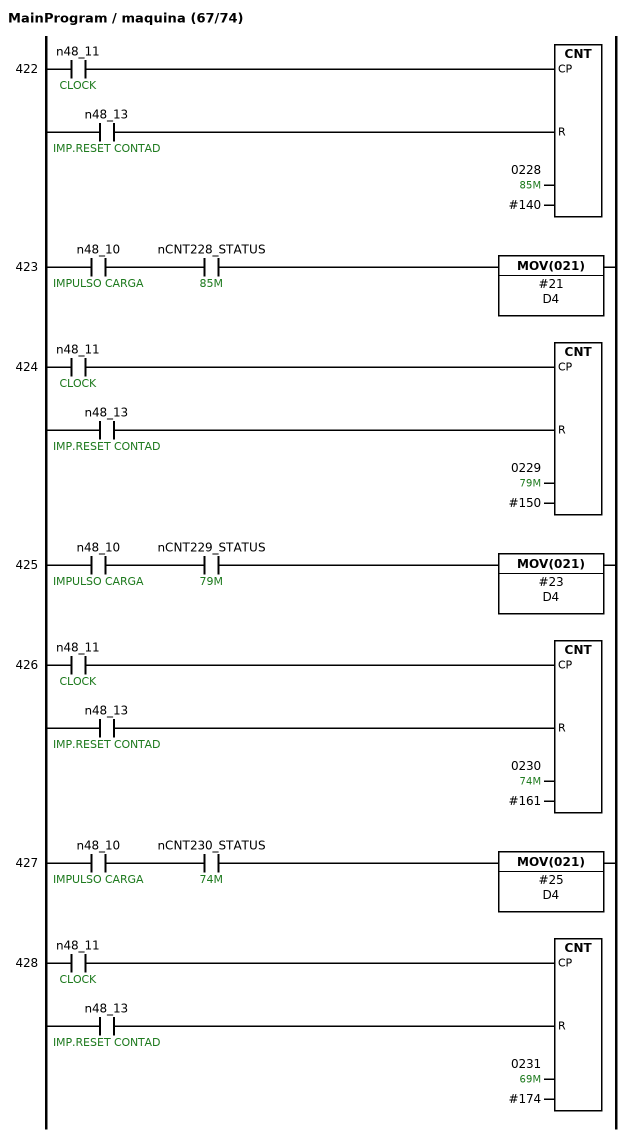
; [picture p72: MainProgram / maquina, rungs 422-428]
; rung 422
LD n48_11  ; CLOCK
LD n48_13  ; IMP.RESET CONTAD
CNT 0228 #140  ; 85M
; rung 423
LD n48_10  ; IMPULSO CARGA
AND nCNT228_STATUS  ; 85M
MOV(021) #21 D4
; rung 424
LD n48_11  ; CLOCK
LD n48_13  ; IMP.RESET CONTAD
CNT 0229 #150  ; 79M
; rung 425
LD n48_10  ; IMPULSO CARGA
AND nCNT229_STATUS  ; 79M
MOV(021) #23 D4
; rung 426
LD n48_11  ; CLOCK
LD n48_13  ; IMP.RESET CONTAD
CNT 0230 #161  ; 74M
; rung 427
LD n48_10  ; IMPULSO CARGA
AND nCNT230_STATUS  ; 74M
MOV(021) #25 D4
; rung 428
LD n48_11  ; CLOCK
LD n48_13  ; IMP.RESET CONTAD
CNT 0231 #174  ; 69M

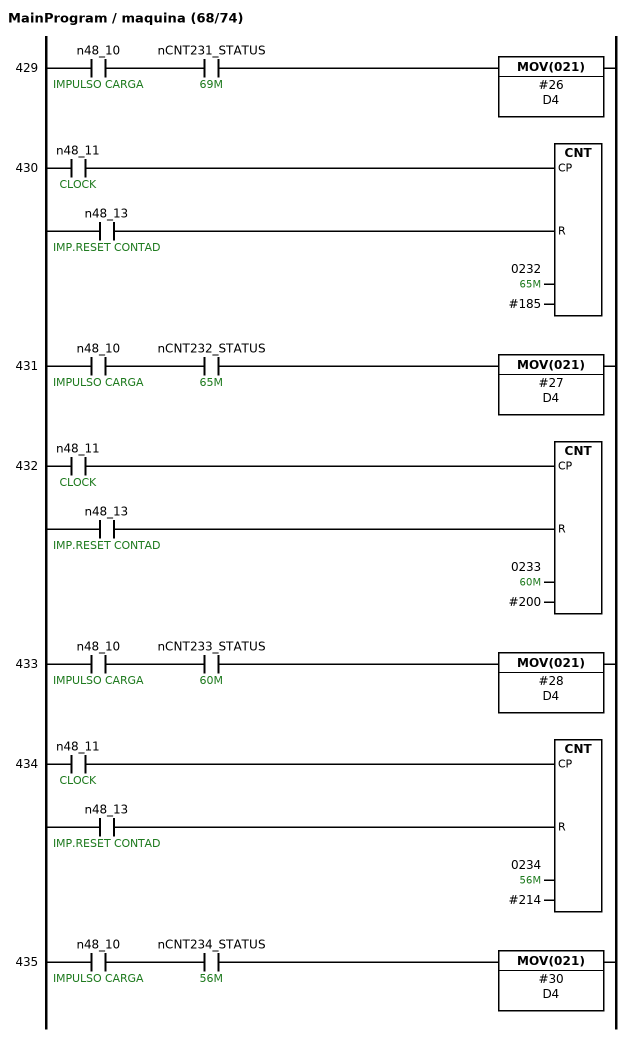
; rung 429
LD n48_10  ; IMPULSO CARGA
AND nCNT231_STATUS  ; 69M
MOV(021) #26 D4
; rung 430
LD n48_11  ; CLOCK
LD n48_13  ; IMP.RESET CONTAD
CNT 0232 #185  ; 65M
; rung 431
LD n48_10  ; IMPULSO CARGA
AND nCNT232_STATUS  ; 65M
MOV(021) #27 D4
; rung 432
LD n48_11  ; CLOCK
LD n48_13  ; IMP.RESET CONTAD
CNT 0233 #200  ; 60M
; rung 433
LD n48_10  ; IMPULSO CARGA
AND nCNT233_STATUS  ; 60M
MOV(021) #28 D4
; rung 434
LD n48_11  ; CLOCK
LD n48_13  ; IMP.RESET CONTAD
CNT 0234 #214  ; 56M
; rung 435
LD n48_10  ; IMPULSO CARGA
AND nCNT234_STATUS  ; 56M
MOV(021) #30 D4

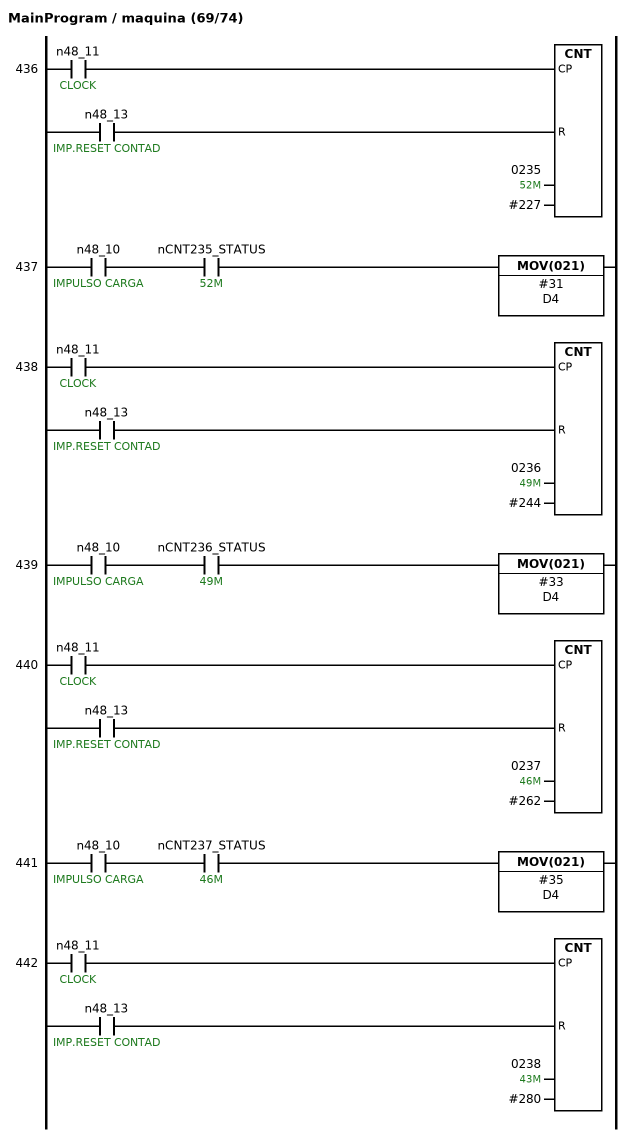
; rung 436
LD n48_11  ; CLOCK
LD n48_13  ; IMP.RESET CONTAD
CNT 0235 #227  ; 52M
; rung 437
LD n48_10  ; IMPULSO CARGA
AND nCNT235_STATUS  ; 52M
MOV(021) #31 D4
; rung 438
LD n48_11  ; CLOCK
LD n48_13  ; IMP.RESET CONTAD
CNT 0236 #244  ; 49M
; rung 439
LD n48_10  ; IMPULSO CARGA
AND nCNT236_STATUS  ; 49M
MOV(021) #33 D4
; rung 440
LD n48_11  ; CLOCK
LD n48_13  ; IMP.RESET CONTAD
CNT 0237 #262  ; 46M
; rung 441
LD n48_10  ; IMPULSO CARGA
AND nCNT237_STATUS  ; 46M
MOV(021) #35 D4
; rung 442
LD n48_11  ; CLOCK
LD n48_13  ; IMP.RESET CONTAD
CNT 0238 #280  ; 43M

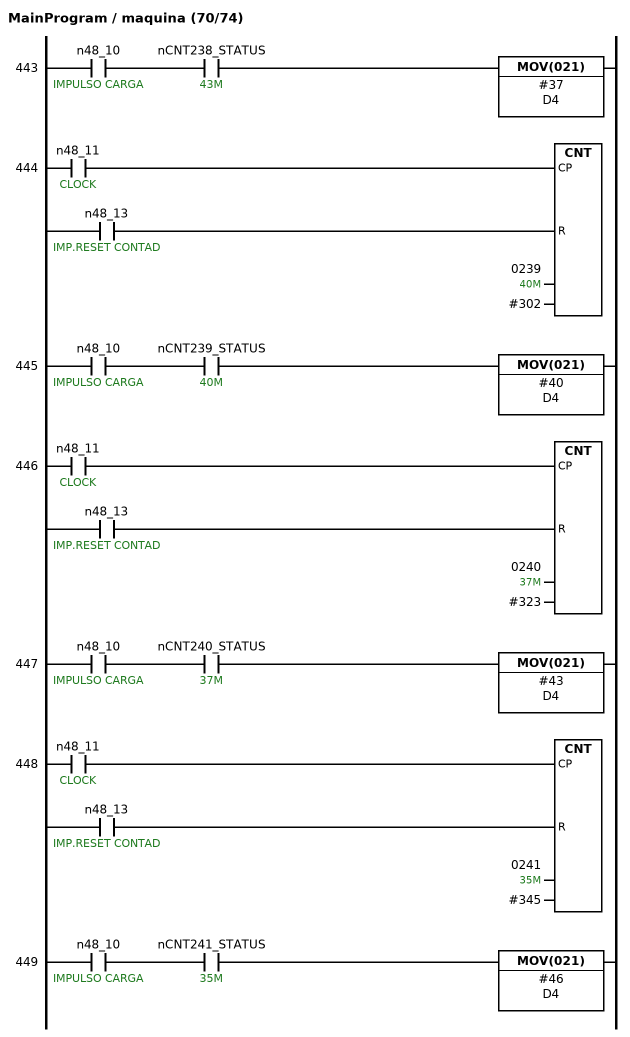
; rung 443
LD n48_10  ; IMPULSO CARGA
AND nCNT238_STATUS  ; 43M
MOV(021) #37 D4
; rung 444
LD n48_11  ; CLOCK
LD n48_13  ; IMP.RESET CONTAD
CNT 0239 #302  ; 40M
; rung 445
LD n48_10  ; IMPULSO CARGA
AND nCNT239_STATUS  ; 40M
MOV(021) #40 D4
; rung 446
LD n48_11  ; CLOCK
LD n48_13  ; IMP.RESET CONTAD
CNT 0240 #323  ; 37M
; rung 447
LD n48_10  ; IMPULSO CARGA
AND nCNT240_STATUS  ; 37M
MOV(021) #43 D4
; rung 448
LD n48_11  ; CLOCK
LD n48_13  ; IMP.RESET CONTAD
CNT 0241 #345  ; 35M
; rung 449
LD n48_10  ; IMPULSO CARGA
AND nCNT241_STATUS  ; 35M
MOV(021) #46 D4

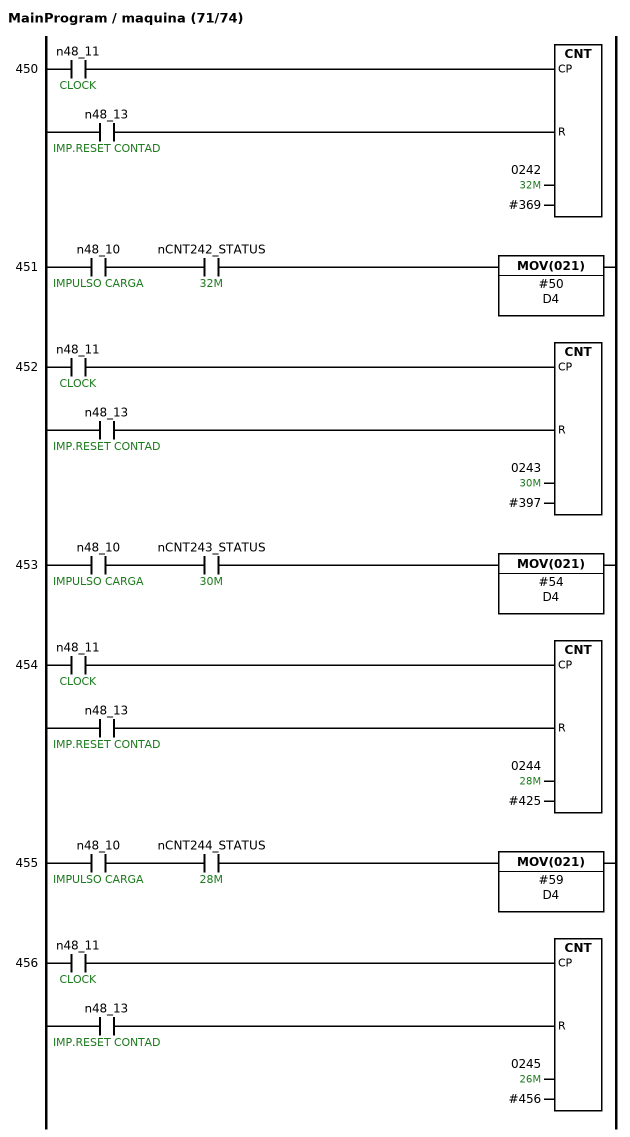
; rung 450
LD n48_11  ; CLOCK
LD n48_13  ; IMP.RESET CONTAD
CNT 0242 #369  ; 32M
; rung 451
LD n48_10  ; IMPULSO CARGA
AND nCNT242_STATUS  ; 32M
MOV(021) #50 D4
; rung 452
LD n48_11  ; CLOCK
LD n48_13  ; IMP.RESET CONTAD
CNT 0243 #397  ; 30M
; rung 453
LD n48_10  ; IMPULSO CARGA
AND nCNT243_STATUS  ; 30M
MOV(021) #54 D4
; rung 454
LD n48_11  ; CLOCK
LD n48_13  ; IMP.RESET CONTAD
CNT 0244 #425  ; 28M
; rung 455
LD n48_10  ; IMPULSO CARGA
AND nCNT244_STATUS  ; 28M
MOV(021) #59 D4
; rung 456
LD n48_11  ; CLOCK
LD n48_13  ; IMP.RESET CONTAD
CNT 0245 #456  ; 26M

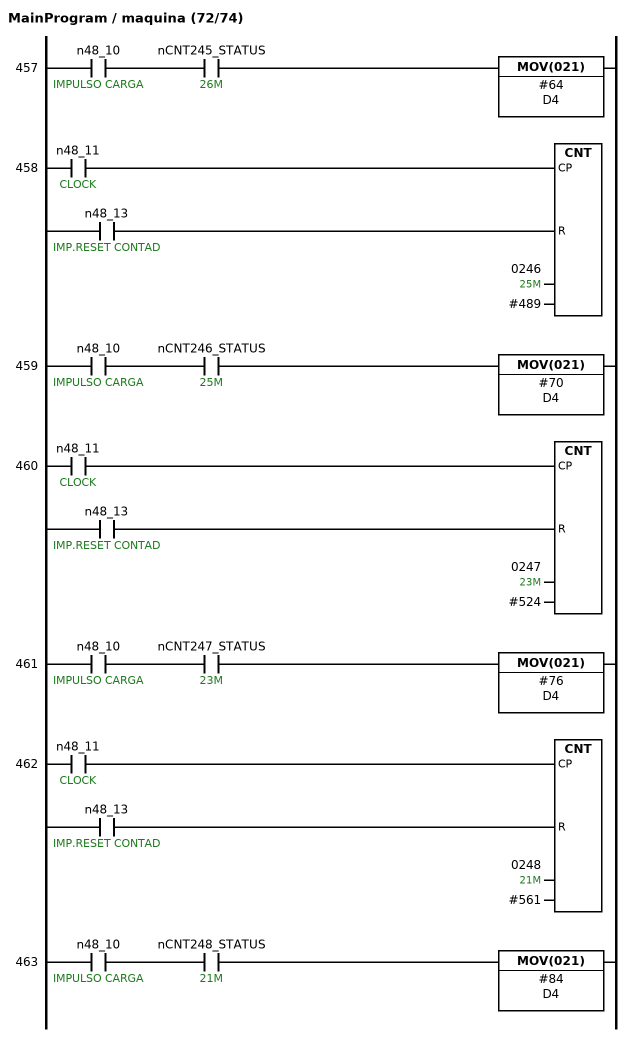
; rung 457
LD n48_10  ; IMPULSO CARGA
AND nCNT245_STATUS  ; 26M
MOV(021) #64 D4
; rung 458
LD n48_11  ; CLOCK
LD n48_13  ; IMP.RESET CONTAD
CNT 0246 #489  ; 25M
; rung 459
LD n48_10  ; IMPULSO CARGA
AND nCNT246_STATUS  ; 25M
MOV(021) #70 D4
; rung 460
LD n48_11  ; CLOCK
LD n48_13  ; IMP.RESET CONTAD
CNT 0247 #524  ; 23M
; rung 461
LD n48_10  ; IMPULSO CARGA
AND nCNT247_STATUS  ; 23M
MOV(021) #76 D4
; rung 462
LD n48_11  ; CLOCK
LD n48_13  ; IMP.RESET CONTAD
CNT 0248 #561  ; 21M
; rung 463
LD n48_10  ; IMPULSO CARGA
AND nCNT248_STATUS  ; 21M
MOV(021) #84 D4

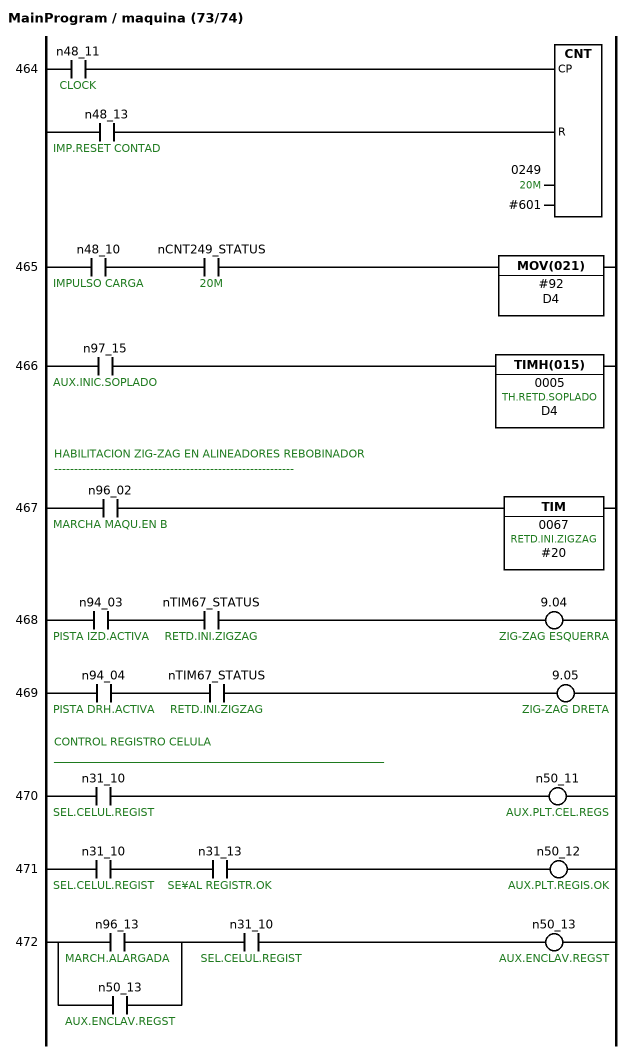
; rung 464
LD n48_11  ; CLOCK
LD n48_13  ; IMP.RESET CONTAD
CNT 0249 #601  ; 20M
; rung 465
LD n48_10  ; IMPULSO CARGA
AND nCNT249_STATUS  ; 20M
MOV(021) #92 D4
; rung 466
LD n97_15  ; AUX.INIC.SOPLADO
TIMH(015) 0005 D4  ; TH.RETD.SOPLADO
; rung 467: HABILITACION ZIG-ZAG EN ALINEADORES REBOBINADOR / ------------------------------------------------------------
LD n96_02  ; MARCHA MAQU.EN B
TIM 0067 #20  ; RETD.INI.ZIGZAG
; rung 468
LD n94_03  ; PISTA IZD.ACTIVA
AND nTIM67_STATUS  ; RETD.INI.ZIGZAG
OUT 9.04  ; ZIG-ZAG ESQUERRA
; rung 469
LD n94_04  ; PISTA DRH.ACTIVA
AND nTIM67_STATUS  ; RETD.INI.ZIGZAG
OUT 9.05  ; ZIG-ZAG DRETA
; rung 470: CONTROL REGISTRO CELULA / ____________________________________________________________
LD n31_10  ; SEL.CELUL.REGIST
OUT n50_11  ; AUX.PLT.CEL.REGS
; rung 471
LD n31_10  ; SEL.CELUL.REGIST
AND n31_13  ; SE¥AL REGISTR.OK
OUT n50_12  ; AUX.PLT.REGIS.OK
; rung 472
LD n96_13  ; MARCH.ALARGADA
OR n50_13  ; AUX.ENCLAV.REGST
AND n31_10  ; SEL.CELUL.REGIST
OUT n50_13  ; AUX.ENCLAV.REGST

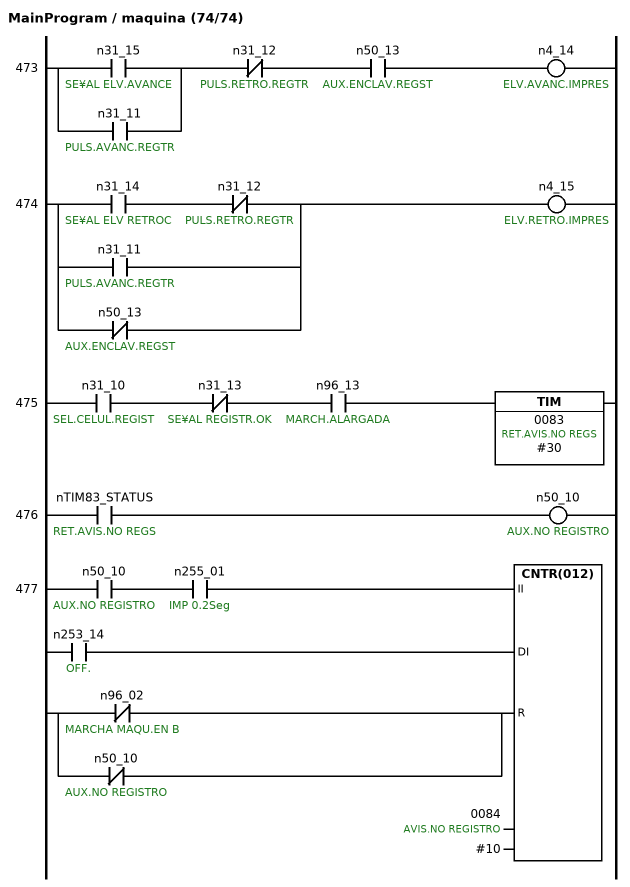
; rung 473
LD n31_15  ; SE¥AL ELV.AVANCE
OR n31_11  ; PULS.AVANC.REGTR
ANDNOT n31_12  ; PULS.RETRO.REGTR
AND n50_13  ; AUX.ENCLAV.REGST
OUT n4_14  ; ELV.AVANC.IMPRES
; rung 474
LD n31_14  ; SE¥AL ELV RETROC
ANDNOT n31_12  ; PULS.RETRO.REGTR
OR n31_11  ; PULS.AVANC.REGTR
ORNOT n50_13  ; AUX.ENCLAV.REGST
OUT n4_15  ; ELV.RETRO.IMPRES
; rung 475
LD n31_10  ; SEL.CELUL.REGIST
ANDNOT n31_13  ; SE¥AL REGISTR.OK
AND n96_13  ; MARCH.ALARGADA
TIM 0083 #30  ; RET.AVIS.NO REGS
; rung 476
LD nTIM83_STATUS  ; RET.AVIS.NO REGS
OUT n50_10  ; AUX.NO REGISTRO
; rung 477
LD n50_10  ; AUX.NO REGISTRO
AND n255_01  ; IMP 0.2Seg
LD n253_14  ; OFF.
LDNOT n96_02  ; MARCHA MAQU.EN B
ORNOT n50_10  ; AUX.NO REGISTRO
CNTR(012) 0084 #10  ; AVIS.NO REGISTRO

### Section Aliniadors

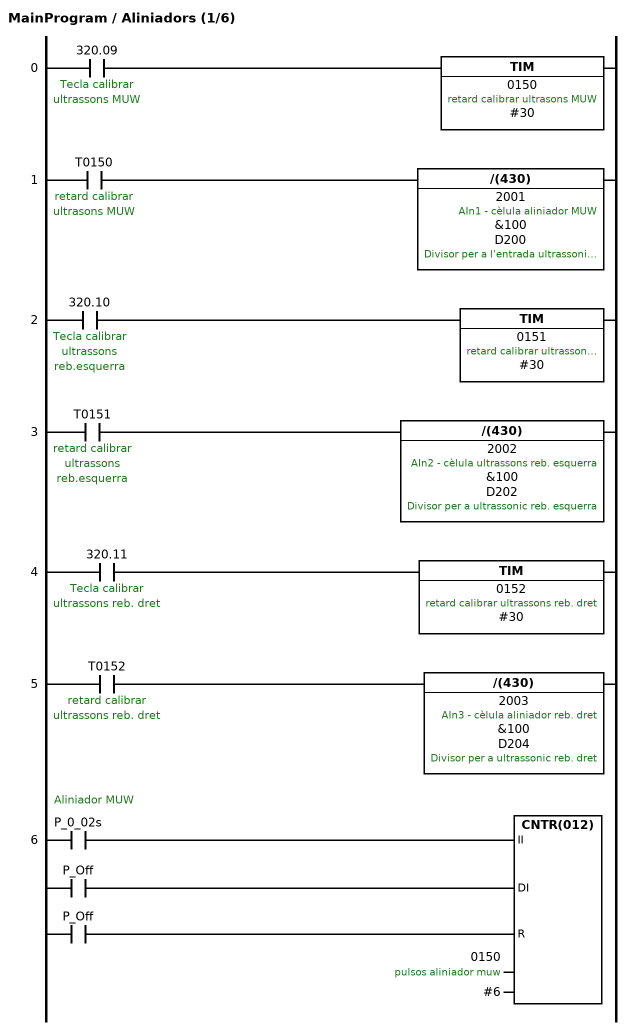
; rung 0
LD 320.09  ; Tecla calibrar ultrassons MUW
TIM 0150 #30  ; retard calibrar ultrasons MUW
; rung 1
LD T0150  ; retard calibrar ultrasons MUW
/(430) 2001 &100 D200  ; AIn1 - cèlula aliniador MUW, Divisor per a l'entrada ultrassonic MUW
; rung 2
LD 320.10  ; Tecla calibrar ultrassons reb.esquerra
TIM 0151 #30  ; retard calibrar ultrassons reb.esquerra
; rung 3
LD T0151  ; retard calibrar ultrassons reb.esquerra
/(430) 2002 &100 D202  ; AIn2 - cèlula ultrassons reb. esquerra, Divisor per a ultrassonic reb. esquerra
; rung 4
LD 320.11  ; Tecla calibrar ultrassons reb. dret
TIM 0152 #30  ; retard calibrar ultrassons reb. dret
; rung 5
LD T0152  ; retard calibrar ultrassons reb. dret
/(430) 2003 &100 D204  ; AIn3 - cèlula aliniador reb. dret, Divisor per a ultrassonic reb. dret
; rung 6: Aliniador MUW
LD P_0_02s
LD P_Off
LD P_Off
CNTR(012) 0150 #6  ; pulsos aliniador muw

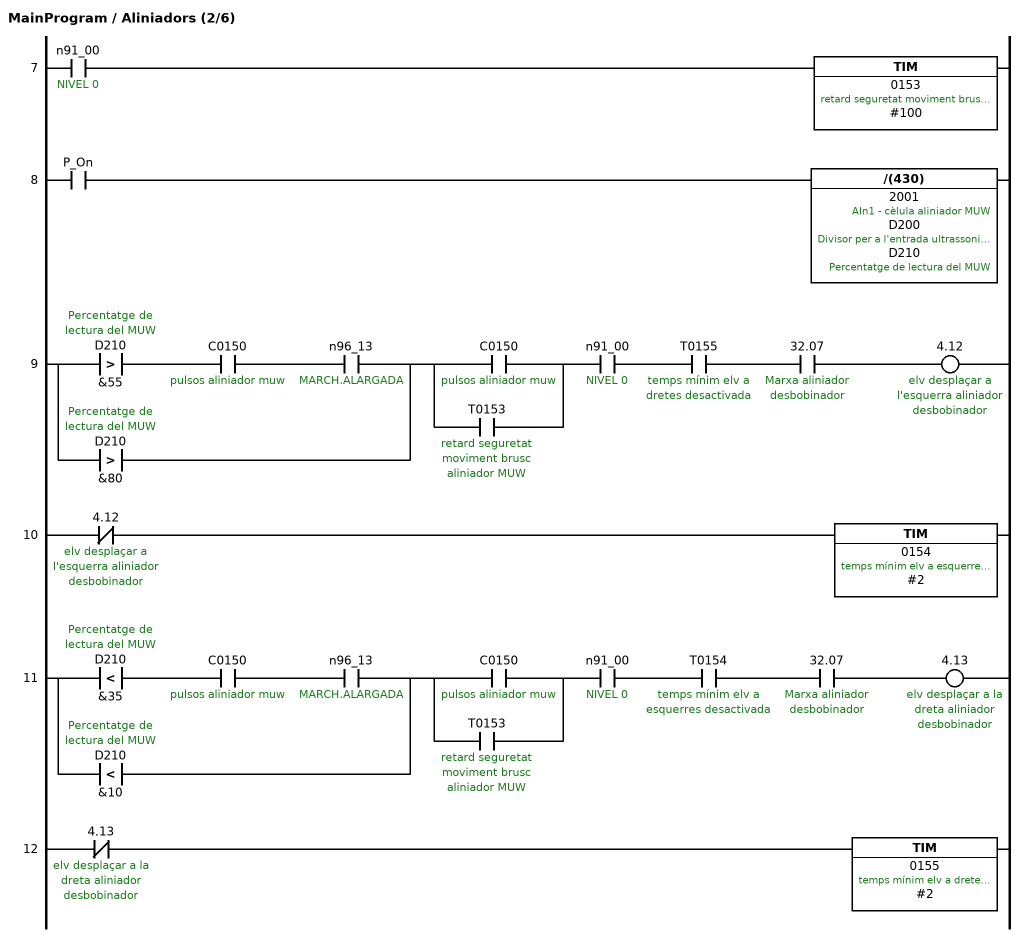
; rung 7
LD n91_00  ; NIVEL 0
TIM 0153 #100  ; retard seguretat moviment brusc aliniador MUW
; rung 8
LD P_On
/(430) 2001 D200 D210  ; AIn1 - cèlula aliniador MUW, Divisor per a l'entrada ultrassonic MUW, Percentatge de lectura del MUW
; rung 9
LD>(320) D210 &55  ; Percentatge de lectura del MUW
AND C0150  ; pulsos aliniador muw
AND n96_13  ; MARCH.ALARGADA
OR>(320) D210 &80  ; Percentatge de lectura del MUW
LD C0150  ; pulsos aliniador muw
OR T0153  ; retard seguretat moviment brusc aliniador MUW
ANDLD
AND n91_00  ; NIVEL 0
AND T0155  ; temps mínim elv a dretes desactivada
AND 32.07  ; Marxa aliniador desbobinador
OUT 4.12  ; elv desplaçar a l'esquerra aliniador desbobinador
; rung 10
LDNOT 4.12  ; elv desplaçar a l'esquerra aliniador desbobinador
TIM 0154 #2  ; temps mínim elv a esquerres desactivada
; rung 11
LD<(310) D210 &35  ; Percentatge de lectura del MUW
AND C0150  ; pulsos aliniador muw
AND n96_13  ; MARCH.ALARGADA
OR<(310) D210 &10  ; Percentatge de lectura del MUW
LD C0150  ; pulsos aliniador muw
OR T0153  ; retard seguretat moviment brusc aliniador MUW
ANDLD
AND n91_00  ; NIVEL 0
AND T0154  ; temps mínim elv a esquerres desactivada
AND 32.07  ; Marxa aliniador desbobinador
OUT 4.13  ; elv desplaçar a la dreta aliniador desbobinador
; rung 12
LDNOT 4.13  ; elv desplaçar a la dreta aliniador desbobinador
TIM 0155 #2  ; temps mínim elv a dretes desactivada

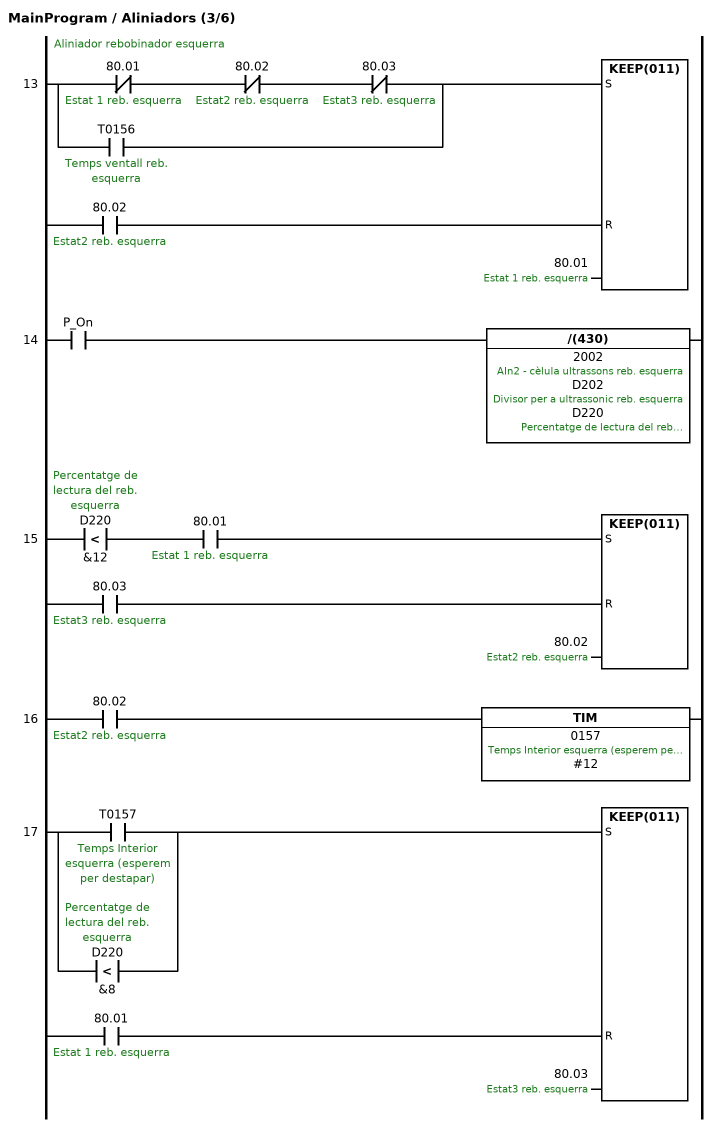
; rung 13: Aliniador rebobinador esquerra
LDNOT 80.01  ; Estat 1 reb. esquerra
ANDNOT 80.02  ; Estat2 reb. esquerra
ANDNOT 80.03  ; Estat3 reb. esquerra
OR T0156  ; Temps ventall reb. esquerra
LD 80.02  ; Estat2 reb. esquerra
KEEP(011) 80.01  ; Estat 1 reb. esquerra
; rung 14
LD P_On
/(430) 2002 D202 D220  ; AIn2 - cèlula ultrassons reb. esquerra, Divisor per a ultrassonic reb. esquerra, Percentatge de lectura del reb. esquerra
; rung 15
LD<(310) D220 &12  ; Percentatge de lectura del reb. esquerra
AND 80.01  ; Estat 1 reb. esquerra
LD 80.03  ; Estat3 reb. esquerra
KEEP(011) 80.02  ; Estat2 reb. esquerra
; rung 16
LD 80.02  ; Estat2 reb. esquerra
TIM 0157 #12  ; Temps Interior esquerra (esperem per destapar)
; rung 17
LD T0157  ; Temps Interior esquerra (esperem per destapar)
OR<(310) D220 &8  ; Percentatge de lectura del reb. esquerra
LD 80.01  ; Estat 1 reb. esquerra
KEEP(011) 80.03  ; Estat3 reb. esquerra

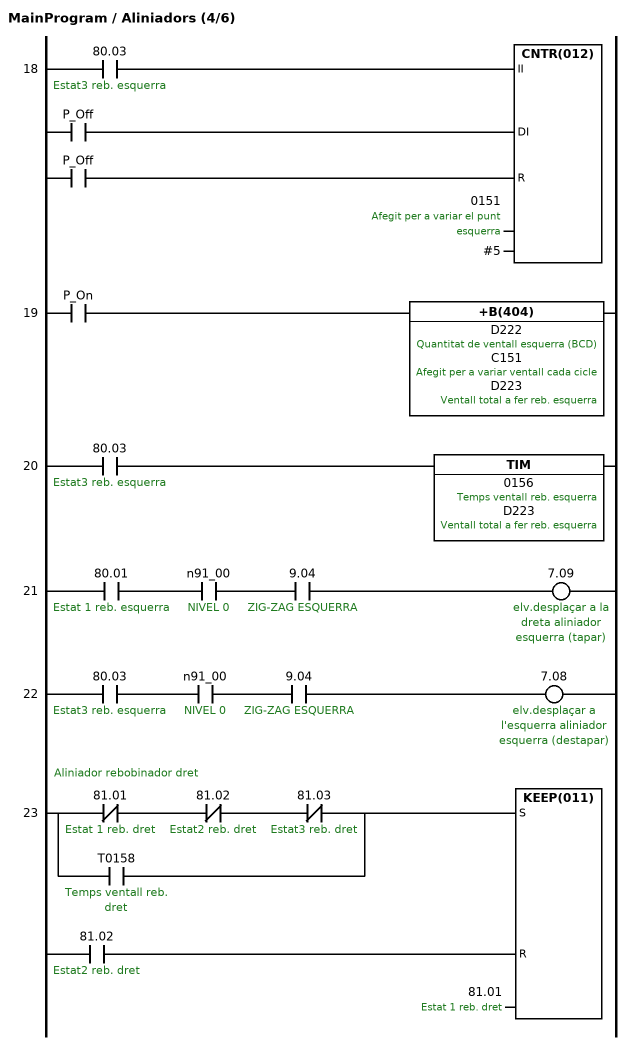
; rung 18
LD 80.03  ; Estat3 reb. esquerra
LD P_Off
LD P_Off
CNTR(012) 0151 #5  ; Afegit per a variar el punt esquerra
; rung 19
LD P_On
+B(404) D222 C151 D223  ; Quantitat de ventall esquerra (BCD), Afegit per a variar ventall cada cicle, Ventall total a fer reb. esquerra
; rung 20
LD 80.03  ; Estat3 reb. esquerra
TIM 0156 D223  ; Ventall total a fer reb. esquerra, Temps ventall reb. esquerra
; rung 21
LD 80.01  ; Estat 1 reb. esquerra
AND n91_00  ; NIVEL 0
AND 9.04  ; ZIG-ZAG ESQUERRA
OUT 7.09  ; elv.desplaçar a la dreta aliniador esquerra (tapar)
; rung 22
LD 80.03  ; Estat3 reb. esquerra
AND n91_00  ; NIVEL 0
AND 9.04  ; ZIG-ZAG ESQUERRA
OUT 7.08  ; elv.desplaçar a l'esquerra aliniador esquerra (destapar)
; rung 23: Aliniador rebobinador dret
LDNOT 81.01  ; Estat 1 reb. dret
ANDNOT 81.02  ; Estat2 reb. dret
ANDNOT 81.03  ; Estat3 reb. dret
OR T0158  ; Temps ventall reb. dret
LD 81.02  ; Estat2 reb. dret
KEEP(011) 81.01  ; Estat 1 reb. dret

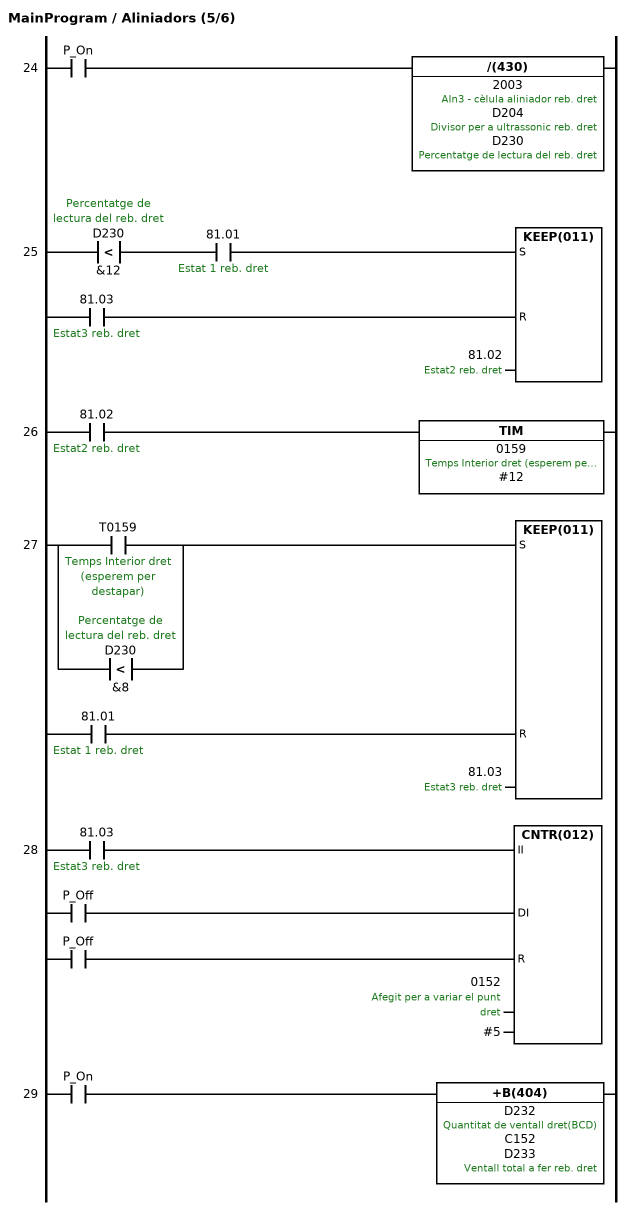
; rung 24
LD P_On
/(430) 2003 D204 D230  ; AIn3 - cèlula aliniador reb. dret, Divisor per a ultrassonic reb. dret, Percentatge de lectura del reb. dret
; rung 25
LD<(310) D230 &12  ; Percentatge de lectura del reb. dret
AND 81.01  ; Estat 1 reb. dret
LD 81.03  ; Estat3 reb. dret
KEEP(011) 81.02  ; Estat2 reb. dret
; rung 26
LD 81.02  ; Estat2 reb. dret
TIM 0159 #12  ; Temps Interior dret (esperem per destapar)
; rung 27
LD T0159  ; Temps Interior dret (esperem per destapar)
OR<(310) D230 &8  ; Percentatge de lectura del reb. dret
LD 81.01  ; Estat 1 reb. dret
KEEP(011) 81.03  ; Estat3 reb. dret
; rung 28
LD 81.03  ; Estat3 reb. dret
LD P_Off
LD P_Off
CNTR(012) 0152 #5  ; Afegit per a variar el punt dret
; rung 29
LD P_On
+B(404) D232 C152 D233  ; Quantitat de ventall dret(BCD), Ventall total a fer reb. dret

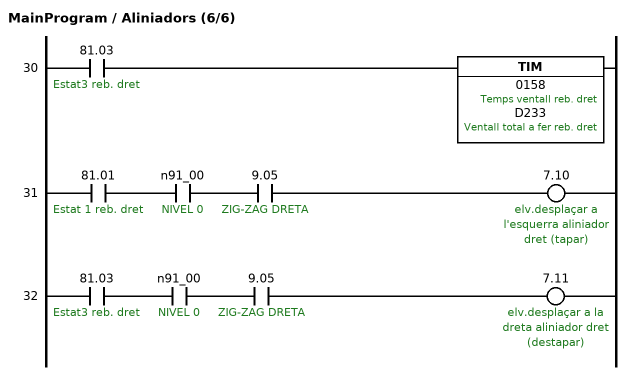
; rung 30
LD 81.03  ; Estat3 reb. dret
TIM 0158 D233  ; Ventall total a fer reb. dret, Temps ventall reb. dret
; rung 31
LD 81.01  ; Estat 1 reb. dret
AND n91_00  ; NIVEL 0
AND 9.05  ; ZIG-ZAG DRETA
OUT 7.10  ; elv.desplaçar a l'esquerra aliniador dret (tapar)
; rung 32
LD 81.03  ; Estat3 reb. dret
AND n91_00  ; NIVEL 0
AND 9.05  ; ZIG-ZAG DRETA
OUT 7.11  ; elv.desplaçar a la dreta aliniador dret (destapar)

### Section HMI

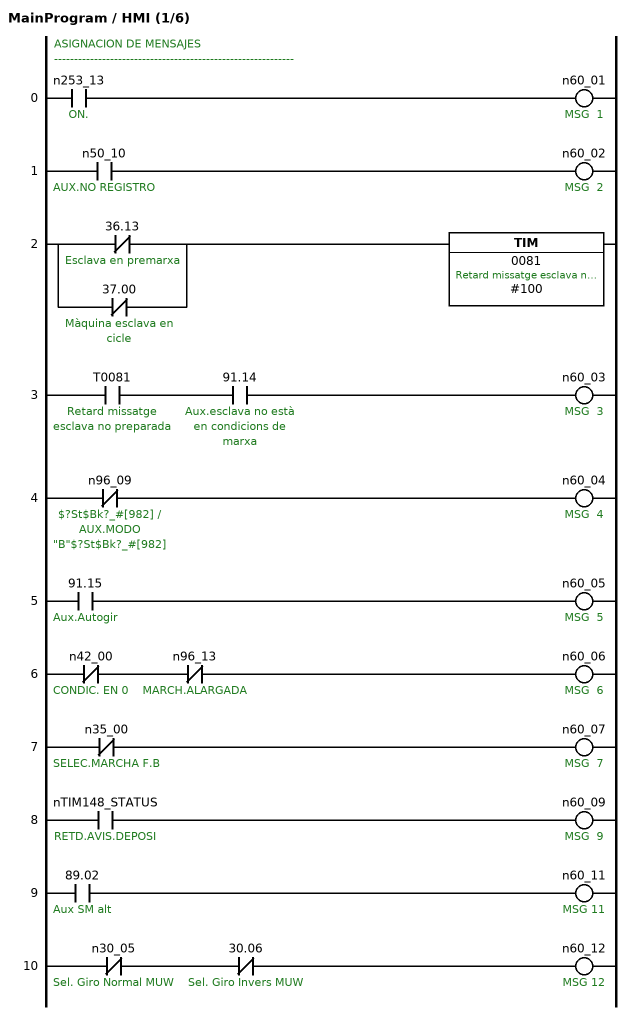
; rung 0: ASIGNACION DE MENSAJES / ------------------------------------------------------------
LD n253_13  ; ON.
OUT n60_01  ; MSG  1
; rung 1
LD n50_10  ; AUX.NO REGISTRO
OUT n60_02  ; MSG  2
; rung 2
LDNOT 36.13  ; Esclava en premarxa
ORNOT 37.00  ; Màquina esclava en cicle
TIM 0081 #100  ; Retard missatge esclava no preparada
; rung 3
LD T0081  ; Retard missatge esclava no preparada
AND 91.14  ; Aux.esclava no està en condicions de marxa
OUT n60_03  ; MSG  3
; rung 4
LDNOT n96_09  ; $?St$Bk?_#[982] / AUX.MODO "B"$?St$Bk?_#[982]
OUT n60_04  ; MSG  4
; rung 5
LD 91.15  ; Aux.Autogir
OUT n60_05  ; MSG  5
; rung 6
LDNOT n42_00  ; CONDIC. EN 0
ANDNOT n96_13  ; MARCH.ALARGADA
OUT n60_06  ; MSG  6
; rung 7
LDNOT n35_00  ; SELEC.MARCHA F.B
OUT n60_07  ; MSG  7
; rung 8
LD nTIM148_STATUS  ; RETD.AVIS.DEPOSI
OUT n60_09  ; MSG  9
; rung 9
LD 89.02  ; Aux SM alt
OUT n60_11  ; MSG 11
; rung 10
LDNOT n30_05  ; Sel. Giro Normal MUW
ANDNOT 30.06  ; Sel. Giro Invers MUW
OUT n60_12  ; MSG 12

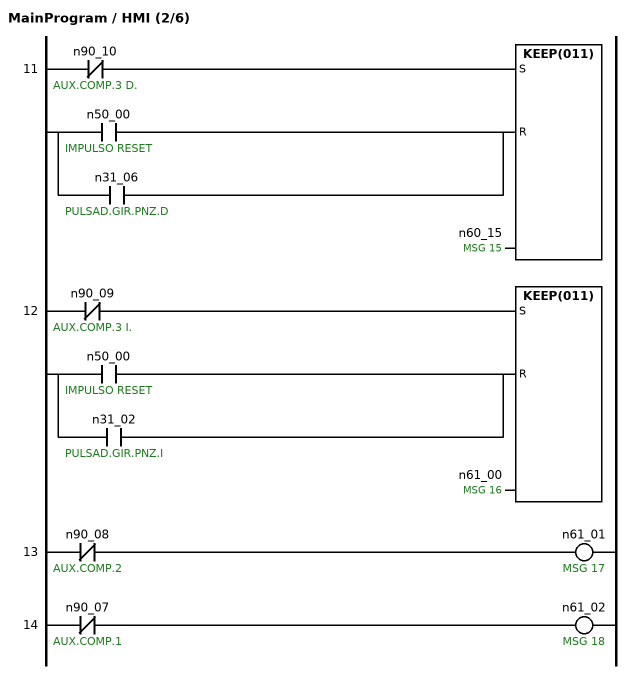
; rung 11
LDNOT n90_10  ; AUX.COMP.3 D.
LD n50_00  ; IMPULSO RESET
OR n31_06  ; PULSAD.GIR.PNZ.D
KEEP(011) n60_15  ; MSG 15
; rung 12
LDNOT n90_09  ; AUX.COMP.3 I.
LD n50_00  ; IMPULSO RESET
OR n31_02  ; PULSAD.GIR.PNZ.I
KEEP(011) n61_00  ; MSG 16
; rung 13
LDNOT n90_08  ; AUX.COMP.2
OUT n61_01  ; MSG 17
; rung 14
LDNOT n90_07  ; AUX.COMP.1
OUT n61_02  ; MSG 18

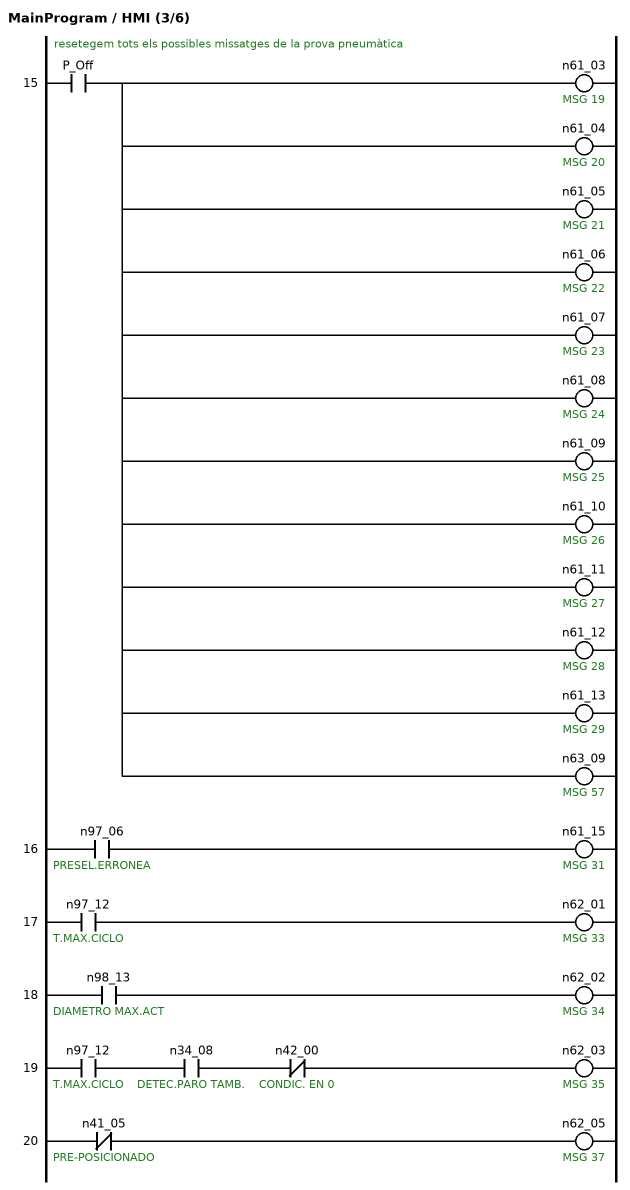
; rung 15: resetegem tots els possibles missatges de la prova pneumàtica
LD P_Off
OUT n61_03  ; MSG 19
OUT n61_04  ; MSG 20
OUT n61_05  ; MSG 21
OUT n61_06  ; MSG 22
OUT n61_07  ; MSG 23
OUT n61_08  ; MSG 24
OUT n61_09  ; MSG 25
OUT n61_10  ; MSG 26
OUT n61_11  ; MSG 27
OUT n61_12  ; MSG 28
OUT n61_13  ; MSG 29
OUT n63_09  ; MSG 57
; rung 16
LD n97_06  ; PRESEL.ERRONEA
OUT n61_15  ; MSG 31
; rung 17
LD n97_12  ; T.MAX.CICLO
OUT n62_01  ; MSG 33
; rung 18
LD n98_13  ; DIAMETRO MAX.ACT
OUT n62_02  ; MSG 34
; rung 19
LD n97_12  ; T.MAX.CICLO
AND n34_08  ; DETEC.PARO TAMB.
ANDNOT n42_00  ; CONDIC. EN 0
OUT n62_03  ; MSG 35
; rung 20
LDNOT n41_05  ; PRE-POSICIONADO
OUT n62_05  ; MSG 37

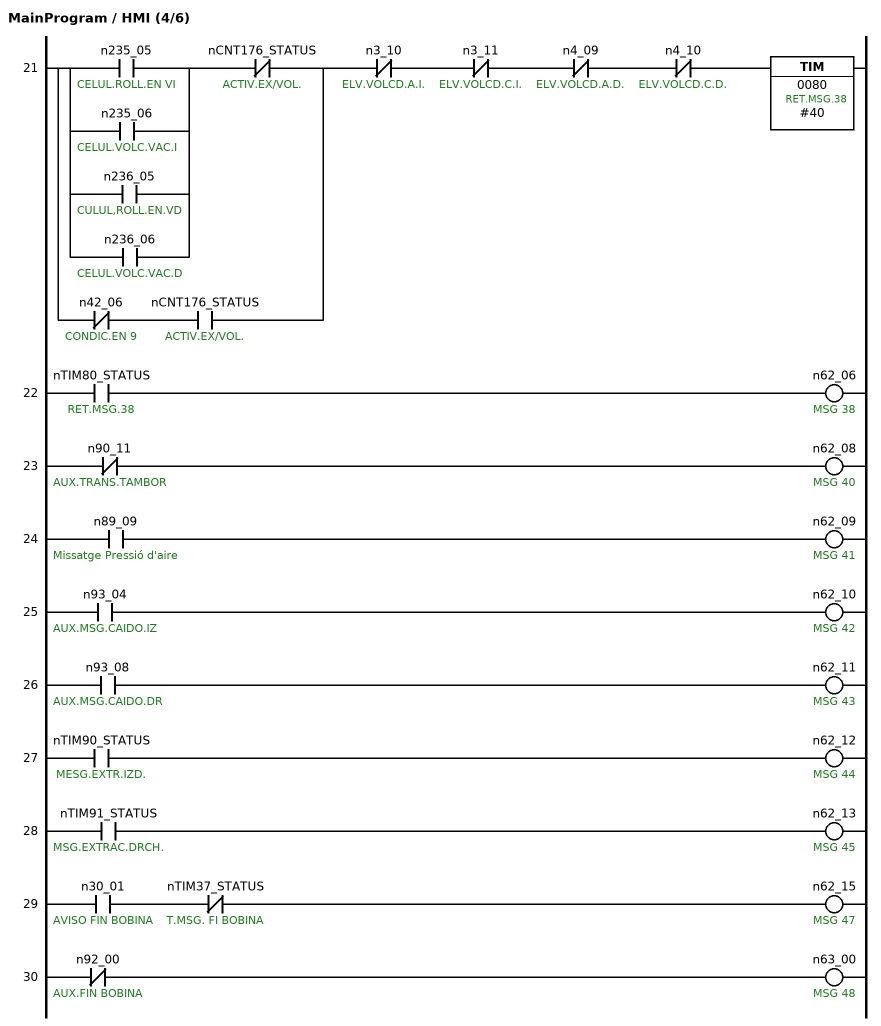
; rung 21
LD n235_05  ; CELUL.ROLL.EN VI
OR n235_06  ; CELUL.VOLC.VAC.I
OR n236_05  ; CULUL,ROLL.EN.VD
OR n236_06  ; CELUL.VOLC.VAC.D
ANDNOT nCNT176_STATUS  ; ACTIV.EX/VOL.
LDNOT n42_06  ; CONDIC.EN 9
AND nCNT176_STATUS  ; ACTIV.EX/VOL.
ORLD
ANDNOT n3_10  ; ELV.VOLCD.A.I.
ANDNOT n3_11  ; ELV.VOLCD.C.I.
ANDNOT n4_09  ; ELV.VOLCD.A.D.
ANDNOT n4_10  ; ELV.VOLCD.C.D.
TIM 0080 #40  ; RET.MSG.38
; rung 22
LD nTIM80_STATUS  ; RET.MSG.38
OUT n62_06  ; MSG 38
; rung 23
LDNOT n90_11  ; AUX.TRANS.TAMBOR
OUT n62_08  ; MSG 40
; rung 24
LD n89_09  ; Missatge Pressió d'aire
OUT n62_09  ; MSG 41
; rung 25
LD n93_04  ; AUX.MSG.CAIDO.IZ
OUT n62_10  ; MSG 42
; rung 26
LD n93_08  ; AUX.MSG.CAIDO.DR
OUT n62_11  ; MSG 43
; rung 27
LD nTIM90_STATUS  ; MESG.EXTR.IZD.
OUT n62_12  ; MSG 44
; rung 28
LD nTIM91_STATUS  ; MSG.EXTRAC.DRCH.
OUT n62_13  ; MSG 45
; rung 29
LD n30_01  ; AVISO FIN BOBINA
ANDNOT nTIM37_STATUS  ; T.MSG. FI BOBINA
OUT n62_15  ; MSG 47
; rung 30
LDNOT n92_00  ; AUX.FIN BOBINA
OUT n63_00  ; MSG 48

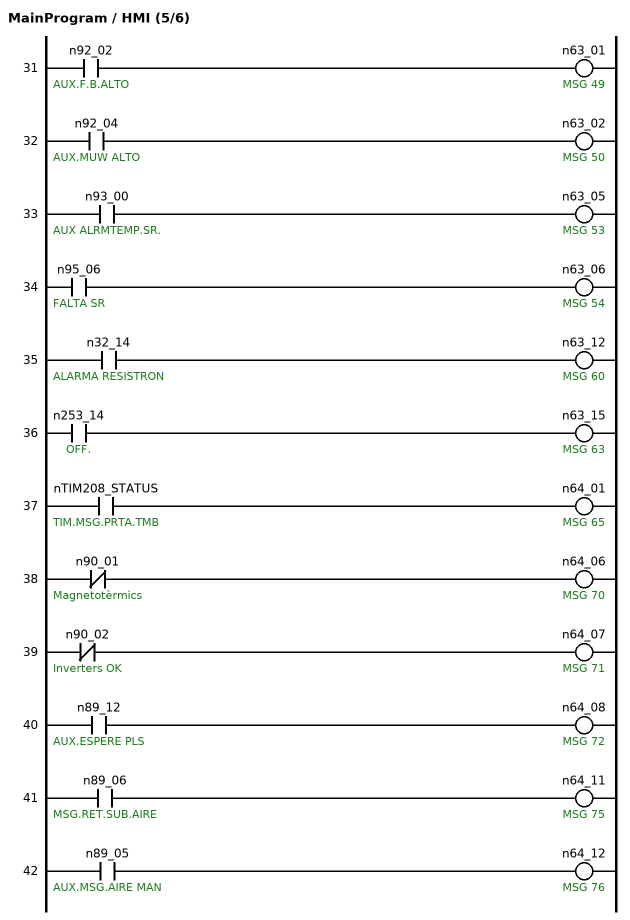
; rung 31
LD n92_02  ; AUX.F.B.ALTO
OUT n63_01  ; MSG 49
; rung 32
LD n92_04  ; AUX.MUW ALTO
OUT n63_02  ; MSG 50
; rung 33
LD n93_00  ; AUX ALRMTEMP.SR.
OUT n63_05  ; MSG 53
; rung 34
LD n95_06  ; FALTA SR
OUT n63_06  ; MSG 54
; rung 35
LD n32_14  ; ALARMA RESISTRON
OUT n63_12  ; MSG 60
; rung 36
LD n253_14  ; OFF.
OUT n63_15  ; MSG 63
; rung 37
LD nTIM208_STATUS  ; TIM.MSG.PRTA.TMB
OUT n64_01  ; MSG 65
; rung 38
LDNOT n90_01  ; Magnetotèrmics
OUT n64_06  ; MSG 70
; rung 39
LDNOT n90_02  ; Inverters OK
OUT n64_07  ; MSG 71
; rung 40
LD n89_12  ; AUX.ESPERE PLS
OUT n64_08  ; MSG 72
; rung 41
LD n89_06  ; MSG.RET.SUB.AIRE
OUT n64_11  ; MSG 75
; rung 42
LD n89_05  ; AUX.MSG.AIRE MAN
OUT n64_12  ; MSG 76

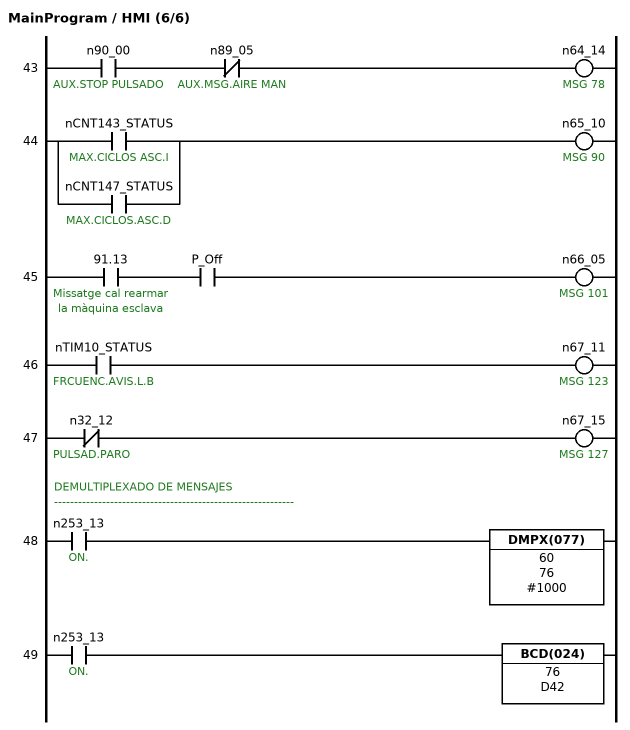
; rung 43
LD n90_00  ; AUX.STOP PULSADO
ANDNOT n89_05  ; AUX.MSG.AIRE MAN
OUT n64_14  ; MSG 78
; rung 44
LD nCNT143_STATUS  ; MAX.CICLOS ASC.I
OR nCNT147_STATUS  ; MAX.CICLOS.ASC.D
OUT n65_10  ; MSG 90
; rung 45
LD 91.13  ; Missatge cal rearmar la màquina esclava
AND P_Off
OUT n66_05  ; MSG 101
; rung 46
LD nTIM10_STATUS  ; FRCUENC.AVIS.L.B
OUT n67_11  ; MSG 123
; rung 47
LDNOT n32_12  ; PULSAD.PARO
OUT n67_15  ; MSG 127
; rung 48: DEMULTIPLEXADO DE MENSAJES / ------------------------------------------------------------
LD n253_13  ; ON.
DMPX(077) 60 76 #1000
; rung 49
LD n253_13  ; ON.
BCD(024) 76 D42

### Section ProvaPneumàtica
; rung 0: SUB PROGRAMA DEDICADO A LAS VERIFICACIONES NEUMATICAS Y DE / CELULAS. DATOS DEL PROGRAMA PRINCIPAL EN EL PASO 2500
; rung 1: ============================================================ / *********   VERIFICACION NEUMATICA Y CELULAS   *************

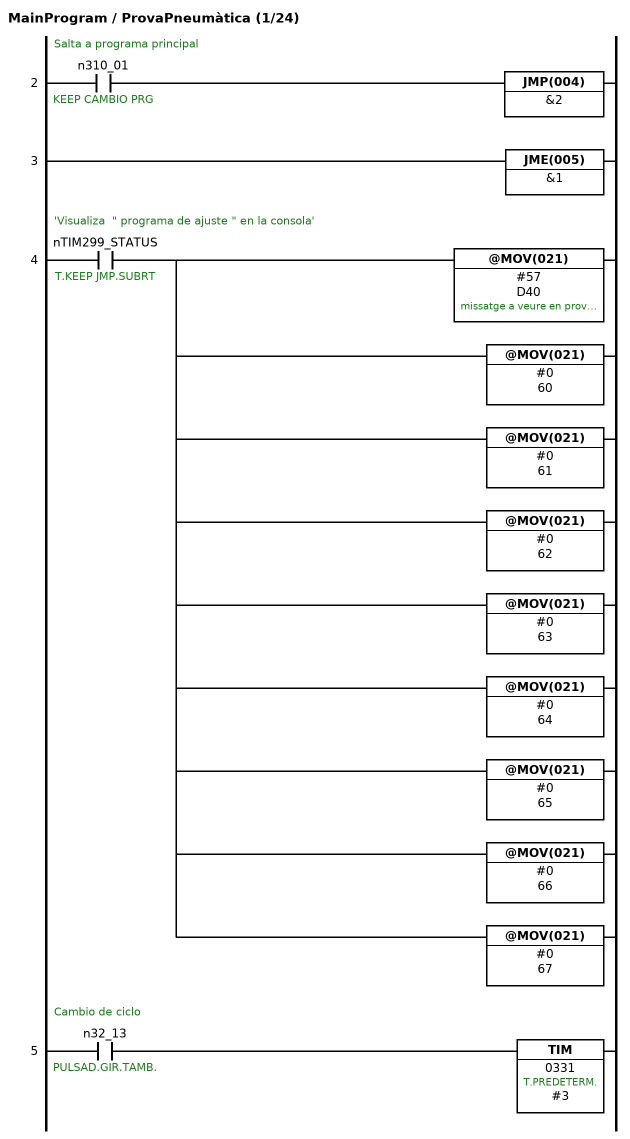
; rung 2: Salta a programa principal
LD n310_01  ; KEEP CAMBIO PRG
JMP(004) &2
; rung 3
JME(005) &1
; rung 4: 'Visualiza  " programa de ajuste " en la consola'
LD nTIM299_STATUS  ; T.KEEP JMP.SUBRT
@MOV(021) #57 D40  ; missatge a veure en prova pneumàtica
@MOV(021) #0 60
@MOV(021) #0 61
@MOV(021) #0 62
@MOV(021) #0 63
@MOV(021) #0 64
@MOV(021) #0 65
@MOV(021) #0 66
@MOV(021) #0 67
; rung 5: Cambio de ciclo
LD n32_13  ; PULSAD.GIR.TAMB.
TIM 0331 #3  ; T.PREDETERM.

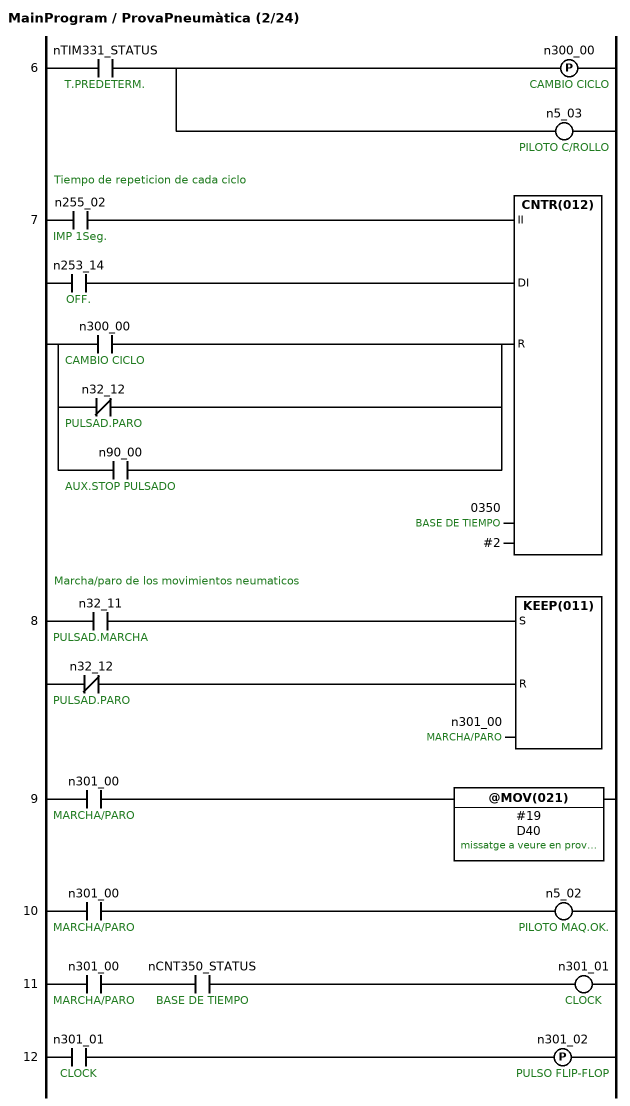
; rung 6
LD nTIM331_STATUS  ; T.PREDETERM.
DIFU(013) n300_00  ; CAMBIO CICLO
OUT n5_03  ; PILOTO C/ROLLO
; rung 7: Tiempo de repeticion de cada ciclo
LD n255_02  ; IMP 1Seg.
LD n253_14  ; OFF.
LD n300_00  ; CAMBIO CICLO
ORNOT n32_12  ; PULSAD.PARO
OR n90_00  ; AUX.STOP PULSADO
CNTR(012) 0350 #2  ; BASE DE TIEMPO
; rung 8: Marcha/paro de los movimientos neumaticos
LD n32_11  ; PULSAD.MARCHA
LDNOT n32_12  ; PULSAD.PARO
KEEP(011) n301_00  ; MARCHA/PARO
; rung 9
LD n301_00  ; MARCHA/PARO
@MOV(021) #19 D40  ; missatge a veure en prova pneumàtica
; rung 10
LD n301_00  ; MARCHA/PARO
OUT n5_02  ; PILOTO MAQ.OK.
; rung 11
LD n301_00  ; MARCHA/PARO
AND nCNT350_STATUS  ; BASE DE TIEMPO
OUT n301_01  ; CLOCK
; rung 12
LD n301_01  ; CLOCK
DIFU(013) n301_02  ; PULSO FLIP-FLOP

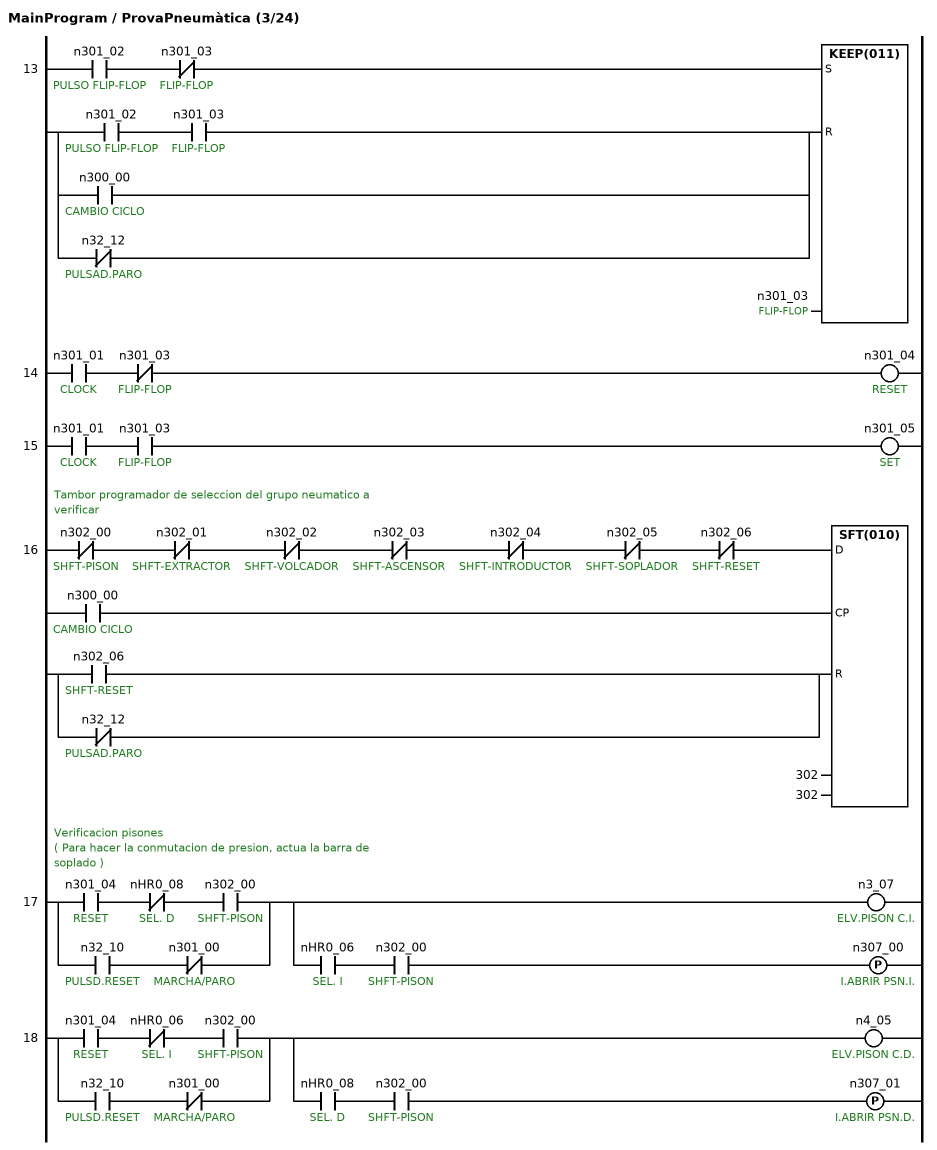
; rung 13
LD n301_02  ; PULSO FLIP-FLOP
ANDNOT n301_03  ; FLIP-FLOP
LD n301_02  ; PULSO FLIP-FLOP
AND n301_03  ; FLIP-FLOP
OR n300_00  ; CAMBIO CICLO
ORNOT n32_12  ; PULSAD.PARO
KEEP(011) n301_03  ; FLIP-FLOP
; rung 14
LD n301_01  ; CLOCK
ANDNOT n301_03  ; FLIP-FLOP
OUT n301_04  ; RESET
; rung 15
LD n301_01  ; CLOCK
AND n301_03  ; FLIP-FLOP
OUT n301_05  ; SET
; rung 16: Tambor programador de seleccion del grupo neumatico a / verificar
LDNOT n302_00  ; SHFT-PISON
ANDNOT n302_01  ; SHFT-EXTRACTOR
ANDNOT n302_02  ; SHFT-VOLCADOR
ANDNOT n302_03  ; SHFT-ASCENSOR
ANDNOT n302_04  ; SHFT-INTRODUCTOR
ANDNOT n302_05  ; SHFT-SOPLADOR
ANDNOT n302_06  ; SHFT-RESET
LD n300_00  ; CAMBIO CICLO
LD n302_06  ; SHFT-RESET
ORNOT n32_12  ; PULSAD.PARO
SFT(010) 302 302
; rung 17: Verificacion pisones / ( Para hacer la conmutacion de presion, actua la barra de / soplado )
LD n301_04  ; RESET
ANDNOT nHR0_08  ; SEL. D
AND n302_00  ; SHFT-PISON
LD n32_10  ; PULSD.RESET
ANDNOT n301_00  ; MARCHA/PARO
ORLD
OUT n3_07  ; ELV.PISON C.I.
AND nHR0_06  ; SEL. I
AND n302_00  ; SHFT-PISON
DIFU(013) n307_00  ; I.ABRIR PSN.I.
; rung 18
LD n301_04  ; RESET
ANDNOT nHR0_06  ; SEL. I
AND n302_00  ; SHFT-PISON
LD n32_10  ; PULSD.RESET
ANDNOT n301_00  ; MARCHA/PARO
ORLD
OUT n4_05  ; ELV.PISON C.D.
AND nHR0_08  ; SEL. D
AND n302_00  ; SHFT-PISON
DIFU(013) n307_01  ; I.ABRIR PSN.D.

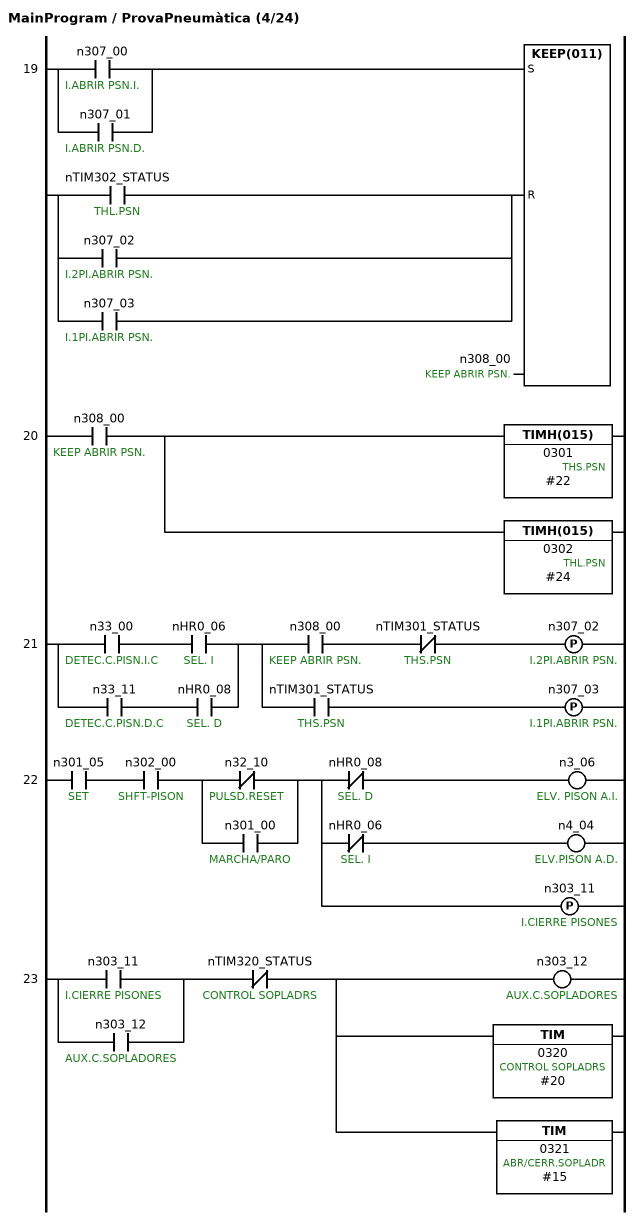
; rung 19
LD n307_00  ; I.ABRIR PSN.I.
OR n307_01  ; I.ABRIR PSN.D.
LD nTIM302_STATUS  ; THL.PSN
OR n307_02  ; I.2PI.ABRIR PSN.
OR n307_03  ; I.1PI.ABRIR PSN.
KEEP(011) n308_00  ; KEEP ABRIR PSN.
; rung 20
LD n308_00  ; KEEP ABRIR PSN.
TIMH(015) 0301 #22  ; THS.PSN
TIMH(015) 0302 #24  ; THL.PSN
; rung 21
LD n33_00  ; DETEC.C.PISN.I.C
AND nHR0_06  ; SEL. I
LD n33_11  ; DETEC.C.PISN.D.C
AND nHR0_08  ; SEL. D
ORLD
OUT TR0
AND n308_00  ; KEEP ABRIR PSN.
ANDNOT nTIM301_STATUS  ; THS.PSN
DIFU(013) n307_02  ; I.2PI.ABRIR PSN.
LD TR0
AND nTIM301_STATUS  ; THS.PSN
DIFU(013) n307_03  ; I.1PI.ABRIR PSN.
; rung 22
LD n301_05  ; SET
AND n302_00  ; SHFT-PISON
LDNOT n32_10  ; PULSD.RESET
OR n301_00  ; MARCHA/PARO
ANDLD
OUT TR0
ANDNOT nHR0_08  ; SEL. D
OUT n3_06  ; ELV. PISON A.I.
LD TR0
ANDNOT nHR0_06  ; SEL. I
OUT n4_04  ; ELV.PISON A.D.
LD TR0
DIFU(013) n303_11  ; I.CIERRE PISONES
; rung 23
LD n303_11  ; I.CIERRE PISONES
OR n303_12  ; AUX.C.SOPLADORES
ANDNOT nTIM320_STATUS  ; CONTROL SOPLADRS
OUT n303_12  ; AUX.C.SOPLADORES
TIM 0320 #20  ; CONTROL SOPLADRS
TIM 0321 #15  ; ABR/CERR.SOPLADR

